PROGRAM Half_Rotation
VAR
	bRotation_Trig : BOOL;
	bFlip_Side: BOOL;
	bProcess: BOOL;
END_VAR

END_PROGRAM

(* stored: Version 1.1.0.1, ProductVersion 3.1.4022.18
   POU Half_Rotation: Id {6ea449ad-6b83-4493-8b59-1e2f14b2084d}, SpecialFunc None *)
